// TwinCAT 3 PLC project UdpDemoPlc
// ProgramVersion: 3.1.4020.1
// libraries:
//   Tc2_Standard, * (Beckhoff Automation GmbH)
//   Tc2_System, * (Beckhoff Automation GmbH)
//   Tc2_Utilities, * (Beckhoff Automation GmbH)
//   Tc3_Module, * (Beckhoff Automation GmbH)
// project tree:
//   DUTs/ receive_data_format.TcDUT, send_data_format.TcDUT, U_IpAdr.TcDUT
//   / PlcTask.TcTTO
//   POUs/ MAIN.TcPOU, FB_UdpReceiver.TcPOU
// real-time tasks:
//   TASK PlcTask: cycle T#1ms, priority 20, ADS port 350
//   TASK PlcTask1: cycle T#1ms, priority 1, ADS port 351
// I/O:
//   DEVICE Device 1 (RT-Ethernet Adapter)

CONFIGURATION UdpDemoPlc
    RESOURCE PLC ON TwinCAT3
        TASK PlcTask(INTERVAL := T#1ms, PRIORITY := 1);
        PROGRAM MAIN WITH PlcTask : MAIN;
    END_RESOURCE
END_CONFIGURATION

// ---- DUTs/receive_data_format.TcDUT
{attribute 'pack_mode' := '0'}
TYPE receive_data_format :
STRUCT
	command		: STRING(4);
	seq_number	: UINT;
	value		: REAL;
END_STRUCT
END_TYPE

// ---- DUTs/send_data_format.TcDUT
{attribute 'pack_mode' := '0'}
TYPE send_data_format :
STRUCT
	command		: STRING(4);
	seq_number	: UINT;
	value		: ULINT;
END_STRUCT
END_TYPE

// ---- DUTs/U_IpAdr.TcDUT
TYPE U_IpAdr :
UNION
	ipAdrInternal : UDINT;
	ipAdr : ARRAY[0..3] OF BYTE;
END_UNION
END_TYPE

// ---- POUs/MAIN.TcPOU
PROGRAM MAIN

VAR
	fbUdp1 : FB_UdpReceiver(nListenPort := 10001);
	send_data		: send_data_format;							// Send message variables
	receive_data 	: receive_data_format;						// Receive message variables
	target_host		: ARRAY [0..3] OF BYTE := [5, 4, 168, 192]; // IP Address of server
	target_port		: UINT := 9998;								// Port number of server listening
	cycle_count		: UINT;
	send_once		: BOOL;
	input_analog_data	AT%I*	: INT;
	parameterized_port		: UINT := 10001;  // Specify receive port by HMI
END_VAR

// 運転中に待ち受けポートを変更したい場合ListenPortプロパティを使って変更する。
fbUdp1.ListenPort := parameterized_port;

// Prepare send data
send_data.command := 'SCOM';
send_data.seq_number := cycle_count;
send_data.value := INT_TO_ULINT(input_analog_data);

IF cycle_count > 65535 THEN
	cycle_count := 0;
ELSE
	cycle_count := cycle_count + 1;
END_IF

// Send request command
IF send_once THEN
	fbUdp1.SendData(
		dest := target_host,
		nTargetPort := target_port,
		data := F_BIGTYPE(pData := ADR(send_data), cbLen := SIZEOF(send_data))
	);
	//send_once := FALSE;
END_IF


fbUdp1(); 

// Get received data to "receive_data" when data received.
IF fbUdp1.receive_complete THEN
	Tc2_System.MEMCPY(ADR(receive_data), fbUdp1.receive_data.pData, fbUdp1.receive_data.cbLen);
END_IF

END_PROGRAM

// ---- POUs/FB_UdpReceiver.TcPOU
{attribute 'c++_compatible'}
FUNCTION_BLOCK FB_UdpReceiver IMPLEMENTS ITcIoUdpProtocolRecv
VAR_INPUT
END_VAR
VAR_OUTPUT
	receive_complete	:BOOL;
	receive_data 		:T_Arg;
END_VAR
VAR
	{attribute 'TcInitSymbol'}
	oid : OTCID; 
	ipUdp : ITcIoUdpProtocol;
	nUdpPort : UINT := 10000;
	nReceivedPakets : UINT;
	uLastReceivedIP : U_IpAdr; 
	hrInit : HRESULT;
	hrSend  : HRESULT;  
	snd_flag	:BOOL;
	ok_counter	:UDINT;
	port_change_counter :UDINT;
END_VAR

IF ipUdp <> 0 THEN
	receive_complete := FALSE;
	ipUdp.CheckReceived();
END_IF

{attribute 'conditionalshow'}
METHOD FB_exit : BOOL
VAR_INPUT
	bInCopyCode : BOOL; // if TRUE, the exit method is called for exiting an instance that is copied afterwards (online change).
END_VAR
IF NOT bInCopyCode THEN // no online change
	IF ipUdp <> 0 THEN 
		ipUdp.UnregisterReceiver(nUdpPort); // Shutdown
		FW_SafeRelease(ADR(ipUdp));
		FB_exit := TRUE; 
	END_IF
END_IF
END_METHOD

{attribute 'conditionalshow'}
METHOD FB_init : BOOL
VAR_INPUT
	bInitRetains : BOOL; // if TRUE, the retain variables are initialized (warm start / cold start)
	bInCopyCode : BOOL;  // if TRUE, the instance afterwards gets moved into the copy code (online change)
	nListenPort: UINT; // Receive port
END_VAR
VAR
	ipSrv : ITComObjectServer;

END_VAR
IF NOT bInCopyCode THEN // no online change
	IF ipUdp = 0 AND oid <> 0 THEN
		IF nListenPort <> 0 THEN
			nUdpPort := nListenPort;
		END_IF
	    hrInit := FW_ObjMgr_GetObjectInstance(	oid:=oid, 
											iid:=TC_GLOBAL_IID_LIST.IID_ITcIoUdpProtocol, 
											pipUnk:=ADR(ipUdp) );
		IF SUCCEEDED(hrInit) THEN 
			IF  SUCCEEDED(ipUdp.RegisterReceiver(nUdpPort, THIS^)) THEN //open port
				FB_init := TRUE;
			ELSE 
				FB_init := FALSE; 
				FW_SafeRelease(ADR(ipUdp));
			END_IF
		END_IF
	ELSIF oid = 0 THEN 
		FB_init := FALSE; 
		hrInit := ERR_INVALID_PARAM; 				
	END_IF
END_IF
END_METHOD

{attribute 'conditionalshow'}
METHOD FB_reinit : BOOL
VAR_INPUT
END_VAR
IF (ipUdp <> 0) THEN 
	ipUdp.RegisterReceiver(nUdpPort, THIS^);
	FB_reinit := TRUE; 
END_IF
END_METHOD

PROPERTY PUBLIC ListenPort : UINT
GET
END_GET
SET
IF nUdpPort = ListenPort THEN
	RETURN;
END_IF

IF SUCCEEDED(ipUdp.UnregisterReceiver(nUdpPort)) THEN
	nUdpPort := ListenPort;
	FB_reinit();
	port_change_counter := port_change_counter + 1;
END_IF
END_SET
END_PROPERTY

{attribute 'object_name' := 'ReceiveData'}
{attribute 'c++_compatible'}
{attribute 'signature_flag' := '33554688'}
{attribute 'pack_mode' := '4'}
{attribute 'show'}
{attribute 'minimal_input_size' := '4'}
METHOD ReceiveData : HRESULT
VAR_INPUT
	ipAddr	: UDINT;
	udpDestPort	: UINT;
	udpSrcPort	: UINT;
	nData	: UDINT;
	pData	: PVOID;
	pVlan	: POINTER TO ETYPE_VLAN_HEADER := 0;
END_VAR
nReceivedPakets := nReceivedPakets+1;
uLastReceivedIP.ipAdrInternal := ipAddr;

IF ipUdp <> 0 THEN
	receive_data.cbLen := nData;
	receive_data.pData := pData;
	receive_complete := TRUE;
END_IF
END_METHOD

METHOD PUBLIC SendData : HRESULT
VAR_INPUT
	dest			: ARRAY [0..3] OF BYTE;
	nTargetPort		: UINT;
	data			: T_ARG;
END_VAR

VAR
	uTargetHostIP	: U_IpAdr;
END_VAR
uTargetHostIP.ipAdr := dest;
hrSend := ipUdp.SendData(uTargetHostIP.ipAdrInternal, nTargetPort, nUdpPort, data.cbLen, data.pData, TRUE, 0); // send data
END_METHOD

{attribute 'object_name' := 'TcAddRef'}
{attribute 'c++_compatible'}
{attribute 'signature_flag' := '33554688'}
{attribute 'pack_mode' := '4'}
{attribute 'show'}
{attribute 'minimal_input_size' := '4'}
METHOD TcAddRef : UDINT
END_METHOD

{attribute 'object_name' := 'TcQueryInterface'}
{attribute 'c++_compatible'}
{attribute 'signature_flag' := '33554688'}
{attribute 'pack_mode' := '4'}
{attribute 'show'}
{attribute 'minimal_input_size' := '4'}
METHOD TcQueryInterface : HRESULT
VAR_INPUT
	iid	: REFERENCE TO IID;
	pipItf	: POINTER TO PVOID;
END_VAR
VAR
	ipUdpRecv : ITcIoUdpProtocolRecv;
	ipUnknown : ITcUnknown;	
END_VAR
IF GuidsEqual(ADR(iid), ADR(TC_GLOBAL_IID_LIST.IID_ITcIoUdpProtocolRecv)) THEN
	ipUdpRecv := THIS^; // cast to interface pointer
	pipItf^ := ITCUNKNOWN_TO_PVOID(ipUdpRecv);
	TcAddRef();
	TcQueryInterface := S_OK;
ELSIF GuidsEqual(ADR(iid), ADR(TC_GLOBAL_IID_LIST.IID_ITcUnknown)) THEN
	ipUnknown := THIS^; // cast to interface pointer
	pipItf^ := ITCUNKNOWN_TO_PVOID(ipUnknown);
	TcAddRef();
	TcQueryInterface := S_OK;
ELSE
	TcQueryInterface := E_HRESULTAdsErr.NOINTERFACE ; //Call super if this fb extends some other
END_IF
END_METHOD

{attribute 'object_name' := 'TcRelease'}
{attribute 'c++_compatible'}
{attribute 'signature_flag' := '33554688'}
{attribute 'pack_mode' := '4'}
{attribute 'show'}
{attribute 'minimal_input_size' := '4'}
METHOD TcRelease : UDINT
END_METHOD

END_FUNCTION_BLOCK
